VAR
	i : INT;
END_VAR
    Rectangle (0,320 64x64), colour toggle: GVL.selectedPieceValidMoveArr[0,4]
        OnMouseClick: execute { GVL.xMoveSpace := 0; GVL.yMoveSpace := 4; }
    Rectangle (64,320 64x64)
    Rectangle (128,320 64x64), colour toggle: GVL.selectedPieceValidMoveArr[2,4]
        OnMouseClick: execute { GVL.xMoveSpace := 2; GVL.yMoveSpace := 4; }
    Rectangle (192,320 64x64)
    Rectangle (0,256 64x64)
    Rectangle (64,256 64x64), colour toggle: GVL.selectedPieceValidMoveArr[1,5]
        OnMouseClick: execute { GVL.xMoveSpace := 1; GVL.yMoveSpace := 5; }
    Rectangle (128,256 64x64)
    Rectangle (192,256 64x64), colour toggle: GVL.selectedPieceValidMoveArr[3,5]
        OnMouseClick: execute { GVL.xMoveSpace := 3; GVL.yMoveSpace := 5; }
    Rectangle (0,192 64x64), colour toggle: GVL.selectedPieceValidMoveArr[0,6]
        OnMouseClick: execute { GVL.xMoveSpace := 0; GVL.yMoveSpace := 6; }
    Rectangle (64,192 64x64)
    Rectangle (128,192 64x64), colour toggle: GVL.selectedPieceValidMoveArr[2,6]
        OnMouseClick: execute { GVL.xMoveSpace := 2; GVL.yMoveSpace := 6; }
    Rectangle (192,192 64x64)
    Rectangle (0,128 64x64)
    Rectangle (192,128 64x64), colour toggle: GVL.selectedPieceValidMoveArr[3,7]
        OnMouseClick: execute { GVL.xMoveSpace := 3; GVL.yMoveSpace := 7; }
    Rectangle (128,128 64x64)
    Rectangle (64,128 64x64), colour toggle: GVL.selectedPieceValidMoveArr[1,7]
        OnMouseClick: execute { GVL.xMoveSpace := 1; GVL.yMoveSpace := 7; }
    Rectangle (256,320 64x64), colour toggle: GVL.selectedPieceValidMoveArr[4,4]
        OnMouseClick: execute { GVL.xMoveSpace := 4; GVL.yMoveSpace := 4; }
    Rectangle (320,320 64x64)
    Rectangle (384,320 64x64), colour toggle: GVL.selectedPieceValidMoveArr[6,4]
        OnMouseClick: execute { GVL.xMoveSpace := 6; GVL.yMoveSpace := 4; }
    Rectangle (448,320 64x64)
    Rectangle (256,256 64x64)
    Rectangle (320,256 64x64), colour toggle: GVL.selectedPieceValidMoveArr[5,5]
        OnMouseClick: execute { GVL.xMoveSpace := 5; GVL.yMoveSpace := 5; }
    Rectangle (384,256 64x64)
    Rectangle (448,256 64x64), colour toggle: GVL.selectedPieceValidMoveArr[7,5]
        OnMouseClick: execute { GVL.xMoveSpace := 7; GVL.yMoveSpace := 5; }
    Rectangle (256,192 64x64), colour toggle: GVL.selectedPieceValidMoveArr[4,6]
        OnMouseClick: execute { GVL.xMoveSpace := 4; GVL.yMoveSpace := 6; }
    Rectangle (320,192 64x64)
    Rectangle (384,192 64x64), colour toggle: GVL.selectedPieceValidMoveArr[6,6]
        OnMouseClick: execute { GVL.xMoveSpace := 6; GVL.yMoveSpace := 6; }
    Rectangle (448,192 64x64)
    Rectangle (256,128 64x64)
    Rectangle (448,128 64x64), colour toggle: GVL.selectedPieceValidMoveArr[7,7]
        OnMouseClick: execute { GVL.xMoveSpace := 7; GVL.yMoveSpace := 7; }
    Rectangle (384,128 64x64)
    Rectangle (320,128 64x64), colour toggle: GVL.selectedPieceValidMoveArr[5,7]
        OnMouseClick: execute { GVL.xMoveSpace := 5; GVL.yMoveSpace := 7; }
    Rectangle (256,576 64x64), colour toggle: GVL.selectedPieceValidMoveArr[4,0]
        OnMouseClick: execute { GVL.xMoveSpace := 4; GVL.yMoveSpace := 0; }
    Rectangle (320,576 64x64)
    Rectangle (384,576 64x64), colour toggle: GVL.selectedPieceValidMoveArr[6,0]
        OnMouseClick: execute { GVL.xMoveSpace := 6; GVL.yMoveSpace := 0; }
    Rectangle (448,576 64x64)
    Rectangle (256,512 64x64)
    Rectangle (320,512 64x64), colour toggle: GVL.selectedPieceValidMoveArr[5,1]
        OnMouseClick: execute { GVL.xMoveSpace := 5; GVL.yMoveSpace := 1; }
    Rectangle (384,512 64x64)
    Rectangle (448,512 64x64), colour toggle: GVL.selectedPieceValidMoveArr[7,1]
        OnMouseClick: execute { GVL.xMoveSpace := 7; GVL.yMoveSpace := 1; }
    Rectangle (256,448 64x64), colour toggle: GVL.selectedPieceValidMoveArr[4,2]
        OnMouseClick: execute { GVL.xMoveSpace := 4; GVL.yMoveSpace := 2; }
    Rectangle (320,448 64x64)
    Rectangle (384,448 64x64), colour toggle: GVL.selectedPieceValidMoveArr[6,2]
        OnMouseClick: execute { GVL.xMoveSpace := 6; GVL.yMoveSpace := 2; }
    Rectangle (448,448 64x64)
    Rectangle (256,384 64x64)
    Rectangle (448,384 64x64), colour toggle: GVL.selectedPieceValidMoveArr[7,3]
        OnMouseClick: execute { GVL.xMoveSpace := 7; GVL.yMoveSpace := 3; }
    Rectangle (384,384 64x64)
    Rectangle (320,384 64x64), colour toggle: GVL.selectedPieceValidMoveArr[5,3]
        OnMouseClick: execute { GVL.xMoveSpace := 5; GVL.yMoveSpace := 3; }
    Rectangle (0,576 64x64), colour toggle: GVL.selectedPieceValidMoveArr[0,0]
        OnMouseClick: execute { GVL.xMoveSpace := 0; GVL.yMoveSpace := 0; }
    Rectangle (64,576 64x64)
    Rectangle (128,576 64x64), colour toggle: GVL.selectedPieceValidMoveArr[2,0]
        OnMouseClick: execute { GVL.xMoveSpace := 2; GVL.yMoveSpace := 0; }
    Rectangle (192,576 64x64)
    Rectangle (0,512 64x64)
    Rectangle (64,512 64x64), colour toggle: GVL.selectedPieceValidMoveArr[1,1]
        OnMouseClick: execute { GVL.xMoveSpace := 1; GVL.yMoveSpace := 1; }
    Rectangle (128,512 64x64)
    Rectangle (192,512 64x64), colour toggle: GVL.selectedPieceValidMoveArr[3,1]
        OnMouseClick: execute { GVL.xMoveSpace := 3; GVL.yMoveSpace := 1; }
    Rectangle (0,448 64x64), colour toggle: GVL.selectedPieceValidMoveArr[0,2]
        OnMouseClick: execute { GVL.xMoveSpace := 0; GVL.yMoveSpace := 2; }
    Rectangle (64,448 64x64)
    Rectangle (128,448 64x64), colour toggle: GVL.selectedPieceValidMoveArr[2,2]
        OnMouseClick: execute { GVL.xMoveSpace := 2; GVL.yMoveSpace := 2; }
    Rectangle (192,448 64x64)
    Rectangle (0,384 64x64)
    Rectangle (192,384 64x64), colour toggle: GVL.selectedPieceValidMoveArr[3,3]
        OnMouseClick: execute { GVL.xMoveSpace := 3; GVL.yMoveSpace := 3; }
    Rectangle (128,384 64x64)
    Rectangle (64,384 64x64), colour toggle: GVL.selectedPieceValidMoveArr[1,3]
        OnMouseClick: execute { GVL.xMoveSpace := 1; GVL.yMoveSpace := 3; }
    Ellipse (256,704 64x64), "%s", text variable: GVL.pieces[0,11].kingText, colour toggle: GVL.pieces[0,11].isSelected
        p3560616238: GVL.pieces[0,11].translatedLocation[0]
        p2738717112: GVL.pieces[0,11].translatedLocation[1]
        OnMouseClick: execute {
            IF(NOT GVL.pieces[0,11].isSelected) THEN
            	// deselect everything
            	FOR i := 0 TO 11 DO
            		GVL.pieces[0,i].isSelected := FALSE;
            		GVL.pieces[1,i].isSelected := FALSE;
            	END_FOR
            	// select the piece
            	GVL.pieces[0,11].isSelected := TRUE;
            	GVL.selectedPieceValidMoveArr := GVL.pieces[0,11].validMoveArr;
            ELSE
            	GVL.pieces[0,11].isSelected := FALSE;
            	GVL.selectedPieceValidMoveArr := GVL.noValidMoveArr;
            END_IF
        }
    Ellipse (256,704 64x64), "%s", text variable: GVL.pieces[0,10].kingText, colour toggle: GVL.pieces[0,10].isSelected
        p3560616238: GVL.pieces[0,10].translatedLocation[0]
        p2738717112: GVL.pieces[0,10].translatedLocation[1]
        OnMouseClick: execute {
            IF(NOT GVL.pieces[0,10].isSelected) THEN
            	// deselect everything
            	FOR i := 0 TO 11 DO
            		GVL.pieces[0,i].isSelected := FALSE;
            		GVL.pieces[1,i].isSelected := FALSE;
            	END_FOR
            	// select the piece
            	GVL.pieces[0,10].isSelected := TRUE;
            	GVL.selectedPieceValidMoveArr := GVL.pieces[0,10].validMoveArr;
            ELSE
            	GVL.pieces[0,10].isSelected := FALSE;
            	GVL.selectedPieceValidMoveArr := GVL.noValidMoveArr;
            END_IF
        }
    Ellipse (128,704 64x64), "%s", text variable: GVL.pieces[0,9].kingText, colour toggle: GVL.pieces[0,9].isSelected
        p3560616238: GVL.pieces[0,9].translatedLocation[0]
        p2738717112: GVL.pieces[0,9].translatedLocation[1]
        OnMouseClick: execute {
            IF(NOT GVL.pieces[0,9].isSelected) THEN
            	// deselect everything
            	FOR i := 0 TO 11 DO
            		GVL.pieces[0,i].isSelected := FALSE;
            		GVL.pieces[1,i].isSelected := FALSE;
            	END_FOR
            	// select the piece
            	GVL.pieces[0,9].isSelected := TRUE;
            	GVL.selectedPieceValidMoveArr := GVL.pieces[0,9].validMoveArr;
            ELSE
            	GVL.pieces[0,9].isSelected := FALSE;
            	GVL.selectedPieceValidMoveArr := GVL.noValidMoveArr;
            END_IF
        }
    Ellipse (128,704 64x64), "%s", text variable: GVL.pieces[0,8].kingText, colour toggle: GVL.pieces[0,8].isSelected
        p3560616238: GVL.pieces[0,8].translatedLocation[0]
        p2738717112: GVL.pieces[0,8].translatedLocation[1]
        OnMouseClick: execute {
            IF(NOT GVL.pieces[0,8].isSelected) THEN
            	// deselect everything
            	FOR i := 0 TO 11 DO
            		GVL.pieces[0,i].isSelected := FALSE;
            		GVL.pieces[1,i].isSelected := FALSE;
            	END_FOR
            	// select the piece
            	GVL.pieces[0,8].isSelected := TRUE;
            	GVL.selectedPieceValidMoveArr := GVL.pieces[0,8].validMoveArr;
            ELSE
            	GVL.pieces[0,8].isSelected := FALSE;
            	GVL.selectedPieceValidMoveArr := GVL.noValidMoveArr;
            END_IF
        }
    Ellipse (128,704 64x64), "%s", text variable: GVL.pieces[0,7].kingText, colour toggle: GVL.pieces[0,7].isSelected
        p3560616238: GVL.pieces[0,7].translatedLocation[0]
        p2738717112: GVL.pieces[0,7].translatedLocation[1]
        OnMouseClick: execute {
            IF(NOT GVL.pieces[0,7].isSelected) THEN
            	// deselect everything
            	FOR i := 0 TO 11 DO
            		GVL.pieces[0,i].isSelected := FALSE;
            		GVL.pieces[1,i].isSelected := FALSE;
            	END_FOR
            	// select the piece
            	GVL.pieces[0,7].isSelected := TRUE;
            	GVL.selectedPieceValidMoveArr := GVL.pieces[0,7].validMoveArr;
            ELSE
            	GVL.pieces[0,7].isSelected := FALSE;
            	GVL.selectedPieceValidMoveArr := GVL.noValidMoveArr;
            END_IF
        }
    Ellipse (128,704 64x64), "%s", text variable: GVL.pieces[0,6].kingText, colour toggle: GVL.pieces[0,6].isSelected
        p3560616238: GVL.pieces[0,6].translatedLocation[0]
        p2738717112: GVL.pieces[0,6].translatedLocation[1]
        OnMouseClick: execute {
            IF(NOT GVL.pieces[0,6].isSelected) THEN
            	// deselect everything
            	FOR i := 0 TO 11 DO
            		GVL.pieces[0,i].isSelected := FALSE;
            		GVL.pieces[1,i].isSelected := FALSE;
            	END_FOR
            	// select the piece
            	GVL.pieces[0,6].isSelected := TRUE;
            	GVL.selectedPieceValidMoveArr := GVL.pieces[0,6].validMoveArr;
            ELSE
            	GVL.pieces[0,6].isSelected := FALSE;
            	GVL.selectedPieceValidMoveArr := GVL.noValidMoveArr;
            END_IF
        }
    Ellipse (128,704 64x64), "%s", text variable: GVL.pieces[0,5].kingText, colour toggle: GVL.pieces[0,5].isSelected
        p3560616238: GVL.pieces[0,5].translatedLocation[0]
        p2738717112: GVL.pieces[0,5].translatedLocation[1]
        OnMouseClick: execute {
            IF(NOT GVL.pieces[0,5].isSelected) THEN
            	// deselect everything
            	FOR i := 0 TO 11 DO
            		GVL.pieces[0,i].isSelected := FALSE;
            		GVL.pieces[1,i].isSelected := FALSE;
            	END_FOR
            	// select the piece
            	GVL.pieces[0,5].isSelected := TRUE;
            	GVL.selectedPieceValidMoveArr := GVL.pieces[0,5].validMoveArr;
            ELSE
            	GVL.pieces[0,5].isSelected := FALSE;
            	GVL.selectedPieceValidMoveArr := GVL.noValidMoveArr;
            END_IF
        }
    Ellipse (0,704 64x64), "%s", text variable: GVL.pieces[0,4].kingText, colour toggle: GVL.pieces[0,4].isSelected
        p3560616238: GVL.pieces[0,4].translatedLocation[0]
        p2738717112: GVL.pieces[0,4].translatedLocation[1]
        OnMouseClick: execute {
            IF(NOT GVL.pieces[0,4].isSelected) THEN
            	// deselect everything
            	FOR i := 0 TO 11 DO
            		GVL.pieces[0,i].isSelected := FALSE;
            		GVL.pieces[1,i].isSelected := FALSE;
            	END_FOR
            	// select the piece
            	GVL.pieces[0,4].isSelected := TRUE;
            	GVL.selectedPieceValidMoveArr := GVL.pieces[0,4].validMoveArr;
            ELSE
            	GVL.pieces[0,4].isSelected := FALSE;
            	GVL.selectedPieceValidMoveArr := GVL.noValidMoveArr;
            END_IF
        }
    Ellipse (0,704 64x64), "%s", text variable: GVL.pieces[0,3].kingText, colour toggle: GVL.pieces[0,3].isSelected
        p3560616238: GVL.pieces[0,3].translatedLocation[0]
        p2738717112: GVL.pieces[0,3].translatedLocation[1]
        OnMouseClick: execute {
            IF(NOT GVL.pieces[0,3].isSelected) THEN
            	// deselect everything
            	FOR i := 0 TO 11 DO
            		GVL.pieces[0,i].isSelected := FALSE;
            		GVL.pieces[1,i].isSelected := FALSE;
            	END_FOR
            	// select the piece
            	GVL.pieces[0,3].isSelected := TRUE;
            	GVL.selectedPieceValidMoveArr := GVL.pieces[0,3].validMoveArr;
            ELSE
            	GVL.pieces[0,3].isSelected := FALSE;
            	GVL.selectedPieceValidMoveArr := GVL.noValidMoveArr;
            END_IF
        }
    Ellipse (0,704 64x64), "%s", text variable: GVL.pieces[0,2].kingText, colour toggle: GVL.pieces[0,2].isSelected
        p3560616238: GVL.pieces[0,2].translatedLocation[0]
        p2738717112: GVL.pieces[0,2].translatedLocation[1]
        OnMouseClick: execute {
            IF(NOT GVL.pieces[0,2].isSelected) THEN
            	// deselect everything
            	FOR i := 0 TO 11 DO
            		GVL.pieces[0,i].isSelected := FALSE;
            		GVL.pieces[1,i].isSelected := FALSE;
            	END_FOR
            	// select the piece
            	GVL.pieces[0,2].isSelected := TRUE;
            	GVL.selectedPieceValidMoveArr := GVL.pieces[0,2].validMoveArr;
            ELSE
            	GVL.pieces[0,2].isSelected := FALSE;
            	GVL.selectedPieceValidMoveArr := GVL.noValidMoveArr;
            END_IF
        }
    Ellipse (0,704 64x64), "%s", text variable: GVL.pieces[0,1].kingText, colour toggle: GVL.pieces[0,1].isSelected
        p3560616238: GVL.pieces[0,1].translatedLocation[0]
        p2738717112: GVL.pieces[0,1].translatedLocation[1]
        OnMouseClick: execute {
            IF(NOT GVL.pieces[0,1].isSelected) THEN
            	// deselect everything
            	FOR i := 0 TO 11 DO
            		GVL.pieces[0,i].isSelected := FALSE;
            		GVL.pieces[1,i].isSelected := FALSE;
            	END_FOR
            	// select the piece
            	GVL.pieces[0,1].isSelected := TRUE;
            	GVL.selectedPieceValidMoveArr := GVL.pieces[0,1].validMoveArr;
            ELSE
            	GVL.pieces[0,1].isSelected := FALSE;
            	GVL.selectedPieceValidMoveArr := GVL.noValidMoveArr;
            END_IF
        }
    Ellipse (0,704 64x64), "%s", text variable: GVL.pieces[0,0].kingText, colour toggle: GVL.pieces[0,0].isSelected
        p3560616238: GVL.pieces[0,0].translatedLocation[0]
        p2738717112: GVL.pieces[0,0].translatedLocation[1]
        OnMouseClick: execute {
            IF(NOT GVL.pieces[0,0].isSelected) THEN
            	// deselect everything
            	FOR i := 0 TO 11 DO
            		GVL.pieces[0,i].isSelected := FALSE;
            		GVL.pieces[1,i].isSelected := FALSE;
            	END_FOR
            	// select the piece
            	GVL.pieces[0,0].isSelected := TRUE;
            	GVL.selectedPieceValidMoveArr := GVL.pieces[0,0].validMoveArr;
            ELSE
            	GVL.pieces[0,0].isSelected := FALSE;
            	GVL.selectedPieceValidMoveArr := GVL.noValidMoveArr;
            END_IF
        }
    Ellipse (192,0 64x64), "%s", text variable: GVL.pieces[1,11].kingText, colour toggle: GVL.pieces[1,11].isSelected
        p3560616238: GVL.pieces[1,11].translatedLocation[0]
        p2738717112: GVL.pieces[1,11].translatedLocation[1]
        OnMouseClick: execute {
            IF(NOT GVL.pieces[1,11].isSelected) THEN
            	// deselect everything
            	FOR i := 0 TO 11 DO
            		GVL.pieces[0,i].isSelected := FALSE;
            		GVL.pieces[1,i].isSelected := FALSE;
            	END_FOR
            	// select the piece
            	GVL.pieces[1,11].isSelected := TRUE;
            	GVL.selectedPieceValidMoveArr := GVL.pieces[1,11].validMoveArr;
            ELSE
            	GVL.pieces[1,11].isSelected := FALSE;
            	GVL.selectedPieceValidMoveArr := GVL.noValidMoveArr;
            END_IF
        }
    Ellipse (190,0 64x64), "%s", text variable: GVL.pieces[1,10].kingText, colour toggle: GVL.pieces[1,10].isSelected
        p3560616238: GVL.pieces[1,10].translatedLocation[0]
        p2738717112: GVL.pieces[1,10].translatedLocation[1]
        OnMouseClick: execute {
            IF(NOT GVL.pieces[1,10].isSelected) THEN
            	// deselect everything
            	FOR i := 0 TO 11 DO
            		GVL.pieces[0,i].isSelected := FALSE;
            		GVL.pieces[1,i].isSelected := FALSE;
            	END_FOR
            	// select the piece
            	GVL.pieces[1,10].isSelected := TRUE;
            	GVL.selectedPieceValidMoveArr := GVL.pieces[1,10].validMoveArr;
            ELSE
            	GVL.pieces[1,10].isSelected := FALSE;
            	GVL.selectedPieceValidMoveArr := GVL.noValidMoveArr;
            END_IF
        }
    Ellipse (320,0 64x64), "%s", text variable: GVL.pieces[1,9].kingText, colour toggle: GVL.pieces[1,9].isSelected
        p3560616238: GVL.pieces[1,9].translatedLocation[0]
        p2738717112: GVL.pieces[1,9].translatedLocation[1]
        OnMouseClick: execute {
            IF(NOT GVL.pieces[1,9].isSelected) THEN
            	// deselect everything
            	FOR i := 0 TO 11 DO
            		GVL.pieces[0,i].isSelected := FALSE;
            		GVL.pieces[1,i].isSelected := FALSE;
            	END_FOR
            	// select the piece
            	GVL.pieces[1,9].isSelected := TRUE;
            	GVL.selectedPieceValidMoveArr := GVL.pieces[1,9].validMoveArr;
            ELSE
            	GVL.pieces[1,9].isSelected := FALSE;
            	GVL.selectedPieceValidMoveArr := GVL.noValidMoveArr;
            END_IF
        }
    Ellipse (320,0 64x64), "%s", text variable: GVL.pieces[1,8].kingText, colour toggle: GVL.pieces[1,8].isSelected
        p3560616238: GVL.pieces[1,8].translatedLocation[0]
        p2738717112: GVL.pieces[1,8].translatedLocation[1]
        OnMouseClick: execute {
            IF(NOT GVL.pieces[1,8].isSelected) THEN
            	// deselect everything
            	FOR i := 0 TO 11 DO
            		GVL.pieces[0,i].isSelected := FALSE;
            		GVL.pieces[1,i].isSelected := FALSE;
            	END_FOR
            	// select the piece
            	GVL.pieces[1,8].isSelected := TRUE;
            	GVL.selectedPieceValidMoveArr := GVL.pieces[1,8].validMoveArr;
            ELSE
            	GVL.pieces[1,8].isSelected := FALSE;
            	GVL.selectedPieceValidMoveArr := GVL.noValidMoveArr;
            END_IF
        }
    Ellipse (320,0 64x64), "%s", text variable: GVL.pieces[1,7].kingText, colour toggle: GVL.pieces[1,7].isSelected
        p3560616238: GVL.pieces[1,7].translatedLocation[0]
        p2738717112: GVL.pieces[1,7].translatedLocation[1]
        OnMouseClick: execute {
            IF(NOT GVL.pieces[1,7].isSelected) THEN
            	// deselect everything
            	FOR i := 0 TO 11 DO
            		GVL.pieces[0,i].isSelected := FALSE;
            		GVL.pieces[1,i].isSelected := FALSE;
            	END_FOR
            	// select the piece
            	GVL.pieces[1,7].isSelected := TRUE;
            	GVL.selectedPieceValidMoveArr := GVL.pieces[1,7].validMoveArr;
            ELSE
            	GVL.pieces[1,7].isSelected := FALSE;
            	GVL.selectedPieceValidMoveArr := GVL.noValidMoveArr;
            END_IF
        }
    Ellipse (320,0 64x64), "%s", text variable: GVL.pieces[1,6].kingText, colour toggle: GVL.pieces[1,6].isSelected
        p3560616238: GVL.pieces[1,6].translatedLocation[0]
        p2738717112: GVL.pieces[1,6].translatedLocation[1]
        OnMouseClick: execute {
            IF(NOT GVL.pieces[1,6].isSelected) THEN
            	// deselect everything
            	FOR i := 0 TO 11 DO
            		GVL.pieces[0,i].isSelected := FALSE;
            		GVL.pieces[1,i].isSelected := FALSE;
            	END_FOR
            	// select the piece
            	GVL.pieces[1,6].isSelected := TRUE;
            	GVL.selectedPieceValidMoveArr := GVL.pieces[1,6].validMoveArr;
            ELSE
            	GVL.pieces[1,6].isSelected := FALSE;
            	GVL.selectedPieceValidMoveArr := GVL.noValidMoveArr;
            END_IF
        }
    Ellipse (320,0 64x64), "%s", text variable: GVL.pieces[1,5].kingText, colour toggle: GVL.pieces[1,5].isSelected
        p3560616238: GVL.pieces[1,5].translatedLocation[0]
        p2738717112: GVL.pieces[1,5].translatedLocation[1]
        OnMouseClick: execute {
            IF(NOT GVL.pieces[1,5].isSelected) THEN
            	// deselect everything
            	FOR i := 0 TO 11 DO
            		GVL.pieces[0,i].isSelected := FALSE;
            		GVL.pieces[1,i].isSelected := FALSE;
            	END_FOR
            	// select the piece
            	GVL.pieces[1,5].isSelected := TRUE;
            	GVL.selectedPieceValidMoveArr := GVL.pieces[1,5].validMoveArr;
            ELSE
            	GVL.pieces[1,5].isSelected := FALSE;
            	GVL.selectedPieceValidMoveArr := GVL.noValidMoveArr;
            END_IF
        }
    Ellipse (448,0 64x64), "%s", text variable: GVL.pieces[1,4].kingText, colour toggle: GVL.pieces[1,4].isSelected
        p3560616238: GVL.pieces[1,4].translatedLocation[0]
        p2738717112: GVL.pieces[1,4].translatedLocation[1]
        OnMouseClick: execute {
            IF(NOT GVL.pieces[1,4].isSelected) THEN
            	// deselect everything
            	FOR i := 0 TO 11 DO
            		GVL.pieces[0,i].isSelected := FALSE;
            		GVL.pieces[1,i].isSelected := FALSE;
            	END_FOR
            	// select the piece
            	GVL.pieces[1,4].isSelected := TRUE;
            	GVL.selectedPieceValidMoveArr := GVL.pieces[1,4].validMoveArr;
            ELSE
            	GVL.pieces[1,4].isSelected := FALSE;
            	GVL.selectedPieceValidMoveArr := GVL.noValidMoveArr;
            END_IF
        }
    Ellipse (450,0 64x64), "%s", text variable: GVL.pieces[1,3].kingText, colour toggle: GVL.pieces[1,3].isSelected
        p3560616238: GVL.pieces[1,3].translatedLocation[0]
        p2738717112: GVL.pieces[1,3].translatedLocation[1]
        OnMouseClick: execute {
            IF(NOT GVL.pieces[1,3].isSelected) THEN
            	// deselect everything
            	FOR i := 0 TO 11 DO
            		GVL.pieces[0,i].isSelected := FALSE;
            		GVL.pieces[1,i].isSelected := FALSE;
            	END_FOR
            	// select the piece
            	GVL.pieces[1,3].isSelected := TRUE;
            	GVL.selectedPieceValidMoveArr := GVL.pieces[1,3].validMoveArr;
            ELSE
            	GVL.pieces[1,3].isSelected := FALSE;
            	GVL.selectedPieceValidMoveArr := GVL.noValidMoveArr;
            END_IF
        }
    Ellipse (450,0 64x64), "%s", text variable: GVL.pieces[1,2].kingText, colour toggle: GVL.pieces[1,2].isSelected
        p3560616238: GVL.pieces[1,2].translatedLocation[0]
        p2738717112: GVL.pieces[1,2].translatedLocation[1]
        OnMouseClick: execute {
            IF(NOT GVL.pieces[1,2].isSelected) THEN
            	// deselect everything
            	FOR i := 0 TO 11 DO
            		GVL.pieces[0,i].isSelected := FALSE;
            		GVL.pieces[1,i].isSelected := FALSE;
            	END_FOR
            	// select the piece
            	GVL.pieces[1,2].isSelected := TRUE;
            	GVL.selectedPieceValidMoveArr := GVL.pieces[1,2].validMoveArr;
            ELSE
            	GVL.pieces[1,2].isSelected := FALSE;
            	GVL.selectedPieceValidMoveArr := GVL.noValidMoveArr;
            END_IF
        }
    Ellipse (450,0 64x64), "%s", text variable: GVL.pieces[1,1].kingText, colour toggle: GVL.pieces[1,1].isSelected
        p3560616238: GVL.pieces[1,1].translatedLocation[0]
        p2738717112: GVL.pieces[1,1].translatedLocation[1]
        OnMouseClick: execute {
            IF(NOT GVL.pieces[1,1].isSelected) THEN
            	// deselect everything
            	FOR i := 0 TO 11 DO
            		GVL.pieces[0,i].isSelected := FALSE;
            		GVL.pieces[1,i].isSelected := FALSE;
            	END_FOR
            	// select the piece
            	GVL.pieces[1,1].isSelected := TRUE;
            	GVL.selectedPieceValidMoveArr := GVL.pieces[1,1].validMoveArr;
            ELSE
            	GVL.pieces[1,1].isSelected := FALSE;
            	GVL.selectedPieceValidMoveArr := GVL.noValidMoveArr;
            END_IF
        }
    Ellipse (450,0 64x64), "%s", text variable: GVL.pieces[1,0].kingText, colour toggle: GVL.pieces[1,0].isSelected
        p3560616238: GVL.pieces[1,0].translatedLocation[0]
        p2738717112: GVL.pieces[1,0].translatedLocation[1]
        OnMouseClick: execute {
            IF(NOT GVL.pieces[1,0].isSelected) THEN
            	// deselect everything
            	FOR i := 0 TO 11 DO
            		GVL.pieces[0,i].isSelected := FALSE;
            		GVL.pieces[1,i].isSelected := FALSE;
            	END_FOR
            	// select the piece
            	GVL.pieces[1,0].isSelected := TRUE;
            	GVL.selectedPieceValidMoveArr := GVL.pieces[1,0].validMoveArr;
            ELSE
            	GVL.pieces[1,0].isSelected := FALSE;
            	GVL.selectedPieceValidMoveArr := GVL.noValidMoveArr;
            END_IF
        }
    Button (619,136 192x38), "Setup Board"
        tap Gameplay.commenceSetup
    Button (624,223 192x38), "Switch Turns"
        OnMouseClick:  ToggleVariable=GVL.redsTurn
    Textfield (627,307 192x38), "%d", text variable: GVL.blackPiecesTaken
END_VISUALIZATION

// CODESYS_SoftMotion_Win_V3/Application/Visualizations/Home_Screen
VISUALIZATION Home_Screen  // 2x2
END_VISUALIZATION

// CODESYS_SoftMotion_Win_V3/Application/Visualizations/Loading_Screen
VISUALIZATION Loading_Screen  // 2x2
END_VISUALIZATION

// CODESYS_SoftMotion_Win_V3/Application/Visualizations/InitScreen
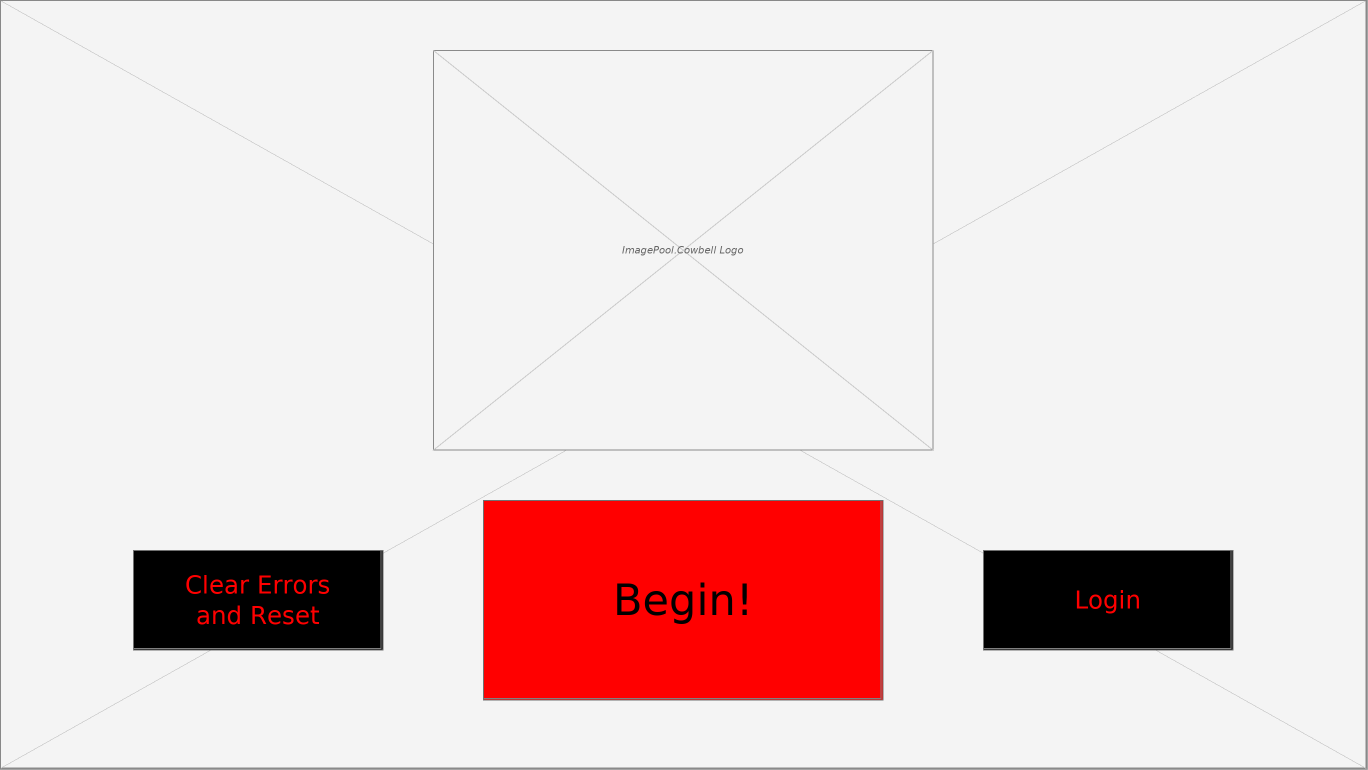
VISUALIZATION InitScreen  // 1368x770
    Image (0,0 1366x768), image: ImagePool.RedCheck
    Image (433,50 500x400), image: ImagePool.Cowbell Logo
    Button (483,500 400x200), "Begin!", text variable: GlobalVars.winnerName
        OnMouseClick:  Assign=MainView, Type=Assignment
        OnMouseClick: execute {
            TestPower.Enable := TRUE;
            JogLogic.startup := TRUE;
            // Run game setup code here
        }
    Button (983,550 250x100), "Login"
        OnMouseClick:  Type=Login
    Button (133,550 250x100), "Clear Errors and Reset"
        OnMouseClick: execute {
            VisuElems.CURRENTLANGUAGE := 'Default';
            JogLogic.startup := TRUE;
            // Any additional resets required to be done here
        }
        OnMouseClick:  Dialog=ErrorsCleared, OpenModal=True, OpenCentered=True
END_VISUALIZATION

// CODESYS_SoftMotion_Win_V3/Application/Visualizations/MainView
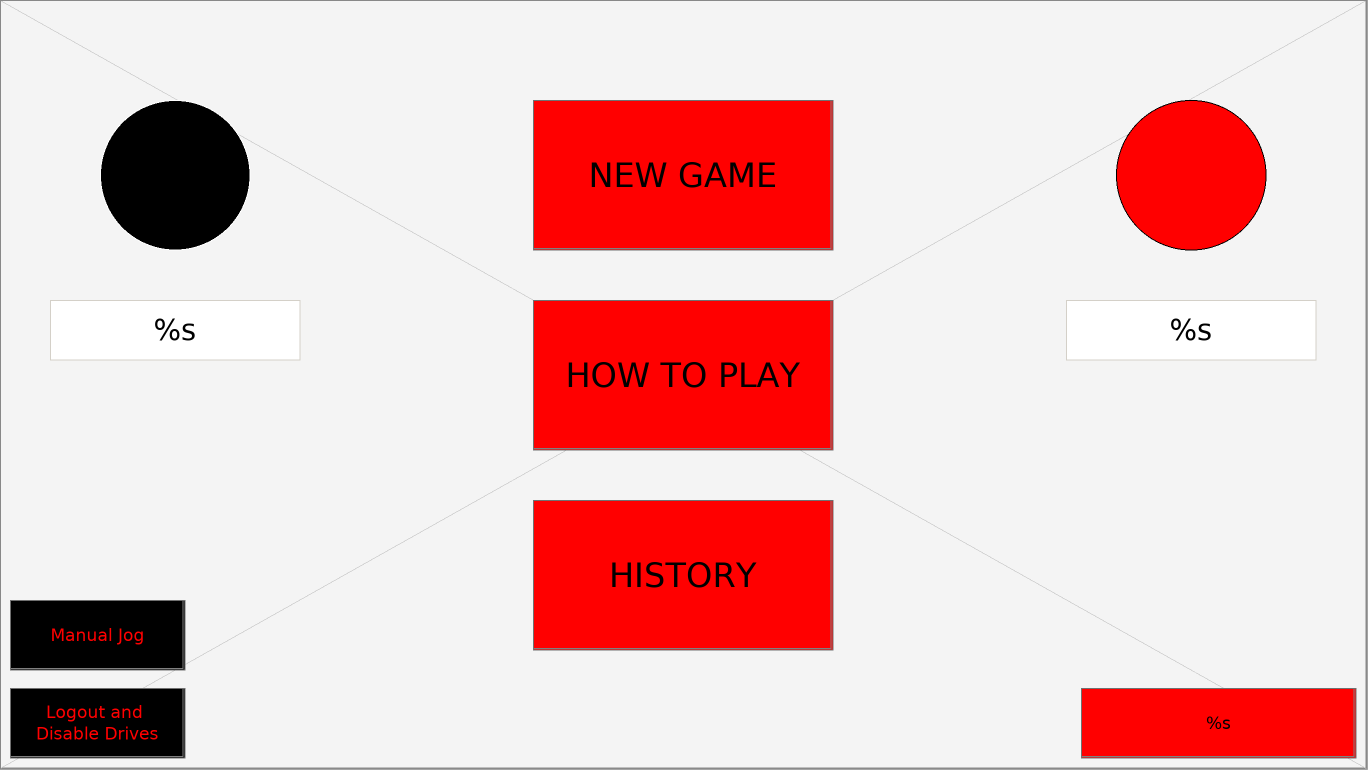
VISUALIZATION MainView  // 1368x770
    Image (0,0 1366x768), image: ImagePool.MedCheck_edited
    Ellipse (100,100 150x150), colour variable: GlobalVars.p1CheckerColor
    Ellipse (1116,100 150x150), colour variable: GlobalVars.p2CheckerColor
    Textfield (50,300 250x60), "%s", text variable: GlobalVars.p1Name
        OnMouseClick: write the text variable via Default
    Textfield (1066,300 250x60), "%s", text variable: GlobalVars.p2Name
        OnMouseClick: write the text variable via Default
    Button (533,100 300x150), "NEW GAME"
        OnMouseClick:  Assign=GameView, Type=Assignment
        OnMouseClick: execute { TestPower.GroupEnable := TRUE; }
    Button (533,300 300x150), "HOW TO PLAY"
        OnMouseClick:  Dialog=HowToPlay, OpenModal=True, OpenCentered=True
    Button (533,500 300x150), "HISTORY"
    Button (10,688 175x70), "Logout and Disable Drives"
        OnMouseClick:  Type=Logout
        OnMouseClick: execute { GlobalVars.systemEnable := FALSE; }
        OnMouseClick:  Assign=InitScreen, Type=Assignment
    Button (10,600 175x70), "Manual Jog"
        OnMouseClick:  Dialog=JogVis, OpenModal=True, OpenCentered=True, PositionX=0, PositionY=0
        OnMouseClick: execute { GlobalVars.systemEnable := TRUE; }
    Button (1081,688 275x70), "%s", text variable: GlobalVars.funnyText
        OnMouseClick: execute {
            GlobalVars.funnyCounter := GlobalVars.funnyCounter + 1;
            IF (GlobalVars.funnyCounter = 1) THEN
            	GlobalVars.funnyText := 'Stop it';
            ELSIF (GlobalVars.funnyCounter = 2) THEN
            	GlobalVars.funnyText := '.........';
            ELSIF (GlobalVars.funnyCounter = 3) THEN
            	GlobalVars.funnyText := 'How would you like it?';
            ELSIF (GlobalVars.funnyCounter = 4) THEN
            	GlobalVars.funnyText := 'Youre only wasting your time';
            ELSIF (GlobalVars.funnyCounter = 5) THEN
            	GlobalVars.funnyText := 'You win';
            ELSIF (GlobalVars.funnyCounter = 7) THEN
            	GlobalVars.funnyText := 'You dont give up easily';
            ELSIF (GlobalVars.funnyCounter = 8) THEN
            	GlobalVars.funnyText := 'Prize for your persistance';
            ELSIF (GlobalVars.funnyCounter = 9) THEN
            	GlobalVars.funnyText := 'lol';
            	VisuElems.CURRENTLANGUAGE := 'CowbellChinese';
            END_IF
        }
END_VISUALIZATION

// CODESYS_SoftMotion_Win_V3/Application/Visualizations/GameView
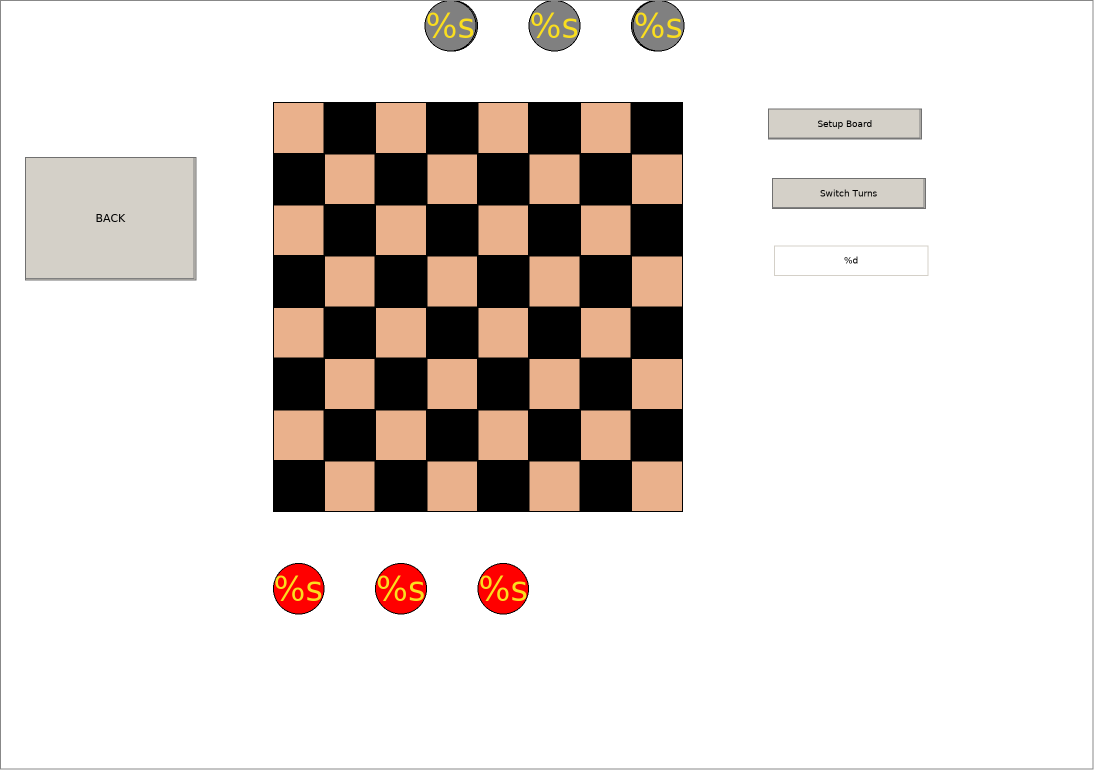
VISUALIZATION GameView  // 1094x770
    Frame (273,0 819x768)
        shows Checkerboard()
    Button (25,157 171x123), "BACK"
        OnMouseClick:  Type=Previous
        OnMouseClick: execute { TestPower.GroupEnable := FALSE; }
END_VISUALIZATION

// CODESYS_SoftMotion_Win_V3/Application/Visualizations/JogVis
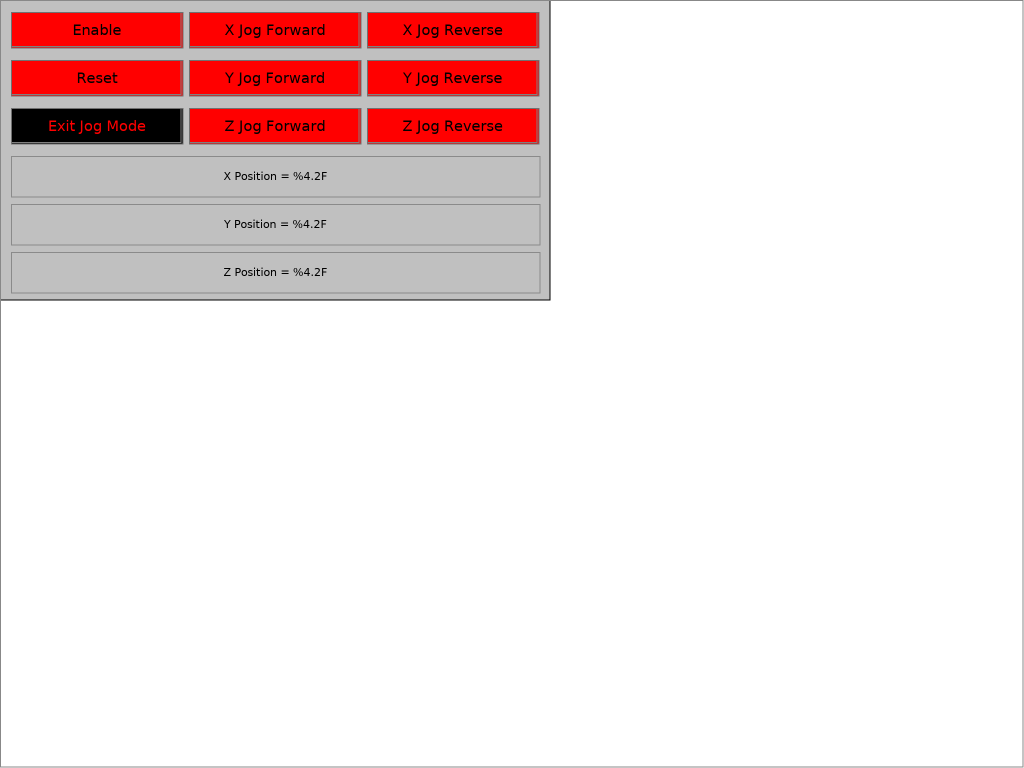
VISUALIZATION JogVis  // 1024x768
    Rectangle (0,0 550x300)
    Button (11,12 172x36), "Enable"
        OnMouseClick:  ToggleVariable=TestPower.Enable
    Button (189,12 172x36), "X Jog Forward"
        tap JogLogic.xJogFwdPressed
    Button (367,12 172x36), "X Jog Reverse"
        tap JogLogic.xJogRevPressed
    Button (189,60 172x36), "Y Jog Forward"
        tap JogLogic.yJogFwdPressed
    Button (367,60 172x36), "Y Jog Reverse"
        tap JogLogic.yJogRevPressed
    Button (11,60 172x36), "Reset"
        OnMouseClick: execute { TestPower.systemReset := TRUE; }
    Button (189,108 172x36), "Z Jog Forward"
        tap JogLogic.zJogFwdPressed
    Button (367,108 172x36), "Z Jog Reverse"
        tap JogLogic.zJogRevPressed
    Frame (11,156 529x41), "X Position = %4.2F", text variable: X.fActPosition
        shows SM3_Basic.LinDrive(m_Input_AXISREF := X)
    Frame (11,204 529x41), "Y Position = %4.2F", text variable: Y.fActPosition
        shows SM3_Basic.LinDrive(m_Input_AXISREF := Y)
    Frame (11,252 529x41), "Z Position = %4.2F", text variable: Z.fActPosition
        shows SM3_Basic.LinDrive(m_Input_AXISREF := Z)
    Button (11,108 172x36), "Exit Jog Mode"
        OnMouseClick:  Dialog=JogVis, Result=OK, NumpadKeypadSet=True
END_VISUALIZATION

// CODESYS_SoftMotion_Win_V3/Application/Visualizations/HowToPlay
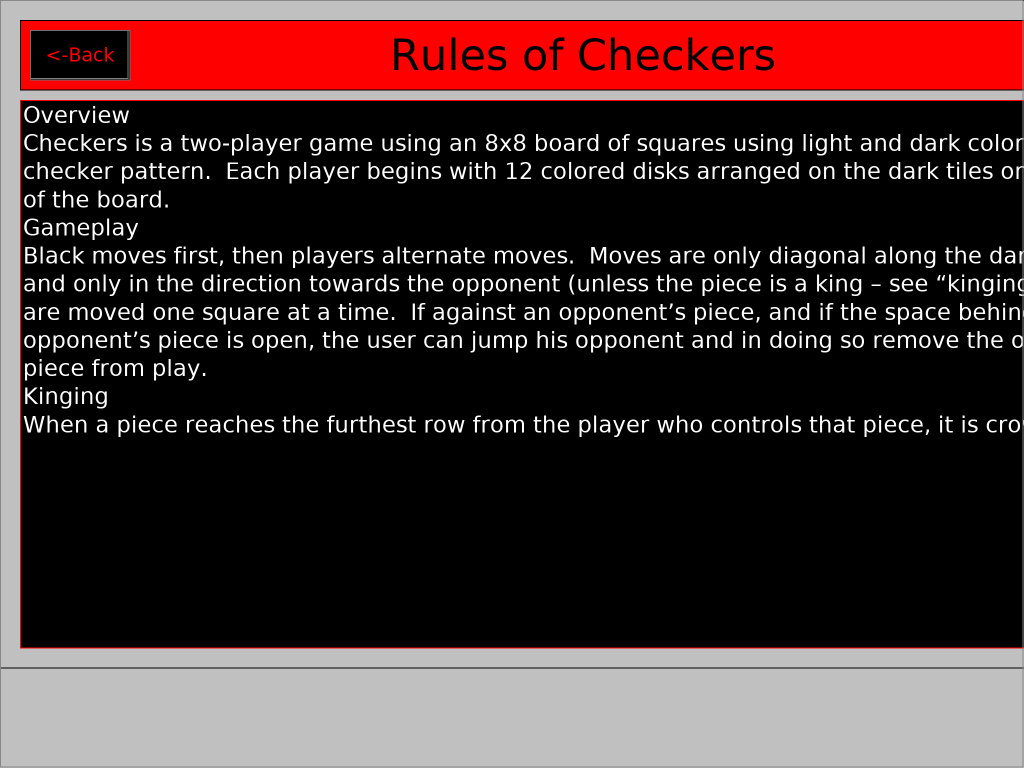
VISUALIZATION HowToPlay  // 1024x768
    Rectangle (0,0 1166x668)
    Textfield (20,100 1126x548), "Overview Checkers is a two-player game using an 8x8 board of squares using light and dark colors in a checker pattern. Each player begins with 12 colored disks arranged on the dark tiles on their side of the board. Gameplay Black moves first, then players alternate moves. Moves are only diagonal along the dark squares and only in the direction towards the opponent (unless the piece is a king – see “kinging”). Pieces are moved one square at a time. If against an opponent’s piece, and if the space behind the opponent’s piece is open, the user can jump his opponent and in doing so remove the opponent piece from play. Kinging When a piece reaches the furthest row from the player who controls that piece, it is crowned and becomes a king. One of the pieces which had been captured is placed on top of the king so that it is twice as high as a single piece. Kings may move both forward and backwards Winning A player wins the game when the opponent cannot make a move. In most cases, this is because all of the opponent's pieces have been captured, but it could also be because all of his pieces are blocked in."
    Textfield (20,20 1126x70), "Rules of Checkers"
    Button (30,30 100x50), "<-Back"
        OnMouseClick:  Dialog=HowToPlay, Result=OK, NumpadKeypadSet=True
END_VISUALIZATION

// CODESYS_SoftMotion_Win_V3/Application/Visualizations/ErrorsCleared
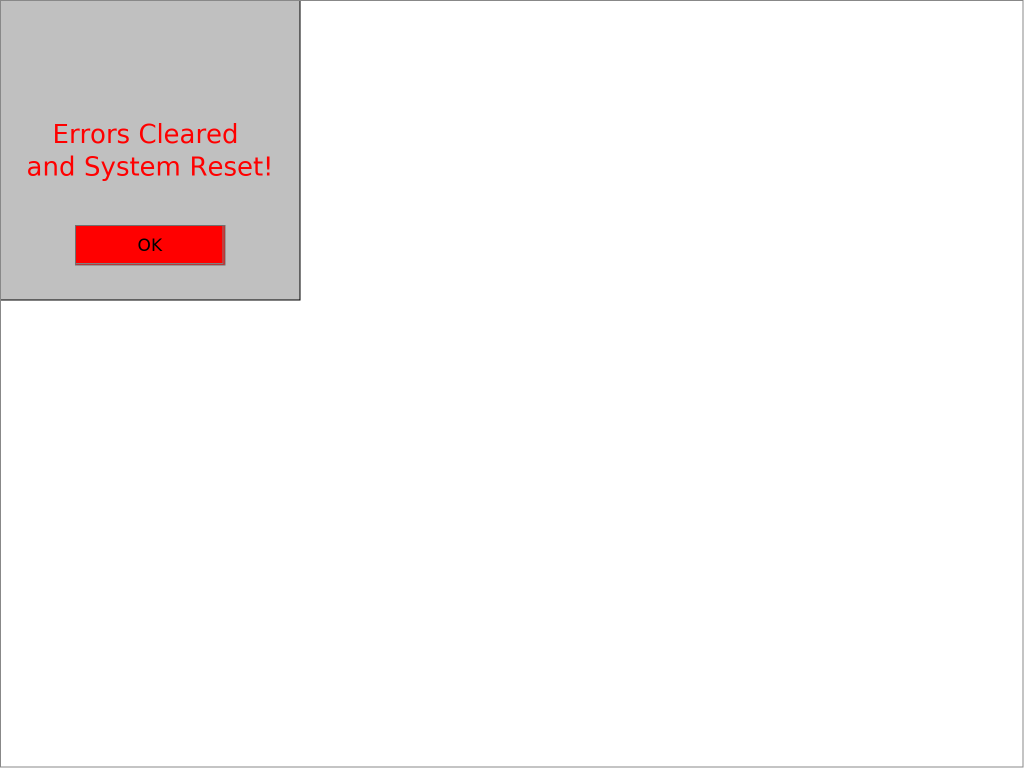
VISUALIZATION ErrorsCleared  // 1024x768
    Rectangle (0,0 300x300), "Errors Cleared and System Reset!"
    Button (75,225 150x40), "OK"
        OnMouseClick:  Dialog=ErrorsCleared, Result=OK, NumpadKeypadSet=True
END_VISUALIZATION

// CODESYS_SoftMotion_Win_V3/Application/Visualizations/Congratulations
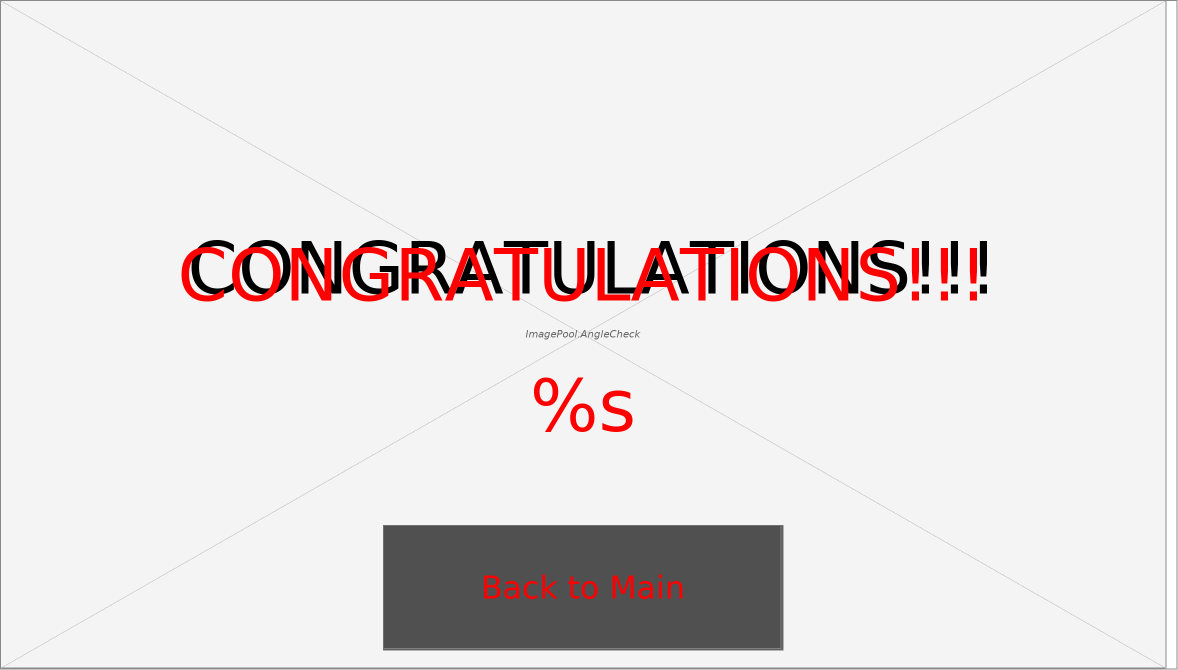
VISUALIZATION Congratulations  // 1178x670
    Image (0,0 1166x668), image: ImagePool.AngleCheck
    Rectangle (10,-7 1166x550), "CONGRATULATIONS!!!"
    Rectangle (0,0 1166x550), "CONGRATULATIONS!!!"
    Button (383,525 400x125), "Back to Main"
    Textfield (0,350 1166x111), "%s", text variable: GlobalVars.winnerName, colour variable: GlobalVars.p2CheckerColor
END_VISUALIZATION

(* text COWBELL_PROGRAMMING_STANDARD
*** General Team Guidelines ***

Program Names (Func, FB, Prog): ProgramName, Program_Name
-Which ever way appears more readable

Variable Names: var1, xVelocity, yVel1
-If global axis variable, axis identifier leads descriptive name.  start lowercase, camelCase

Functions, FunctionBlocks: These should not use global variables, if it can be avoided.  
These types should be able to copy and paste into a new program.

( * Header Comment * ) - good for describing chuncks of code
// In line comment - good for describing a single line

Programs, GlobalVars, etc. will be placed in the POUs so that we can work with the simulator from home.  Don't forget to copy programs to the required task!


Functions can only be called, take inputs and have defined outputs.  Good for math or modifiers.
Function Blocks must be called in a program and do not have explicitly defined inputs and outputs.  Good for repetive chunks of code.  
Programs are the only items that are run in the Task Configuration list.  Programs will call Functions and Function Blocks as required.  

*For Visual Stuff, let's try to stay with the Arial family of Fonts
*)

(* text GameInformation
Logins:

Admin : 1234
Tech : 123
User: play
*)
